{attribute 'qualified_only'}
{attribute 'strict'}
TYPE eSupplyState :
(
	enum_member := 0
);
END_TYPE

(* stored: Version 1.1.0.1, ProductVersion 3.1.4024.12
   DUT eSupplyState: Id {32750b5d-e700-40a3-a03f-af0f0b44efeb} *)
